TYPE unBN_IDM_header_in :
UNION
	bits	: stBN_IDM_header_in;	// bit access
	raw		: BYTE;				// byte access
END_UNION
END_TYPE

(* stored: Version 1.1.0.1, ProductVersion 3.1.4024.6
   DUT unBN_IDM_header_in: Id {7b22c0e8-fe32-446e-85ef-c6452bb428b3} *)
